FUNCTION_BLOCK BoolBindingReadOnlyTest EXTENDS TcUnit.FB_TestSuite
VAR
END_VAR

CheckIsBinded();
BindingReturnsSameValue();
NegatedBindingReturnsNegatedValue();

METHOD BindingReturnsSameValue : BOOL
VAR
	expected : BOOL;
	actual : BOOL;
	
	binding : BoolBindingReadOnly;
	variable : BOOL;
END_VAR
TcUnit.TEST('Binding returns same value');

binding.Bind(variable);

expected := FALSE;
actual := binding.Value;

AssertEquals(
	Expected := expected,
	Actual := actual,
	Message := 'Value should return FALSE if binded variable is FALSE');
	
variable := TRUE;

expected := TRUE;
actual := binding.Value;

AssertEquals(
	Expected := expected,
	Actual := actual,
	Message := 'Value should return TRUE if binded variable is TRUE');

TEST_FINISHED();
END_METHOD

METHOD CheckIsBinded : BOOL
VAR
	expected : BOOL;
	actual : BOOL;
	
	binding : BoolBindingReadOnly;
	variable : BOOL;
END_VAR
TcUnit.TEST('Check binded');

expected := FALSE;
actual := binding.IsBinded;

AssertEquals(
	Expected := expected,
	Actual := actual,
	Message := 'IsBinded should be FALSE before binding');

binding.Bind(variable);

expected := TRUE;
actual := binding.IsBinded;

AssertEquals(
	Expected := expected,
	Actual := actual,
	Message := 'IsBinded should be TRUE after successful Bind()');

TEST_FINISHED();
END_METHOD

METHOD NegatedBindingReturnsNegatedValue : BOOL
VAR
	expected : BOOL;
	actual : BOOL;
	
	binding : BoolBindingReadOnly;
	variable : BOOL;
END_VAR
TcUnit.TEST('Negated binding returns negated value');

binding.Bind(variable);
binding.Negate := TRUE;

expected := TRUE;
actual := binding.Value;

AssertEquals(
	Expected := expected,
	Actual := actual,
	Message := 'Value should return TRUE if binded variable is FALSE');
	
variable := TRUE;

expected := FALSE;
actual := binding.Value;

AssertEquals(
	Expected := expected,
	Actual := actual,
	Message := 'Value should return FALSE if binded variable is TRUE');

TEST_FINISHED();
END_METHOD

END_FUNCTION_BLOCK

(* stored: Version 1.1.0.1, ProductVersion 3.1.4024.12
   POU BoolBindingReadOnlyTest: Id {5ec9cc84-43d1-04b3-01a2-75e05e6f1483}, SpecialFunc None
   Method BindingReturnsSameValue: Id {7e0fd542-12ee-098a-03d0-bcdfeb50173b}
   Method CheckIsBinded: Id {06675ca2-ed9f-0a59-218c-8044f4d3ab81}
   Method NegatedBindingReturnsNegatedValue: Id {5b70dafd-2432-09ad-3235-d008d9be7557} *)
